SUBAPPLICATION mapping_Uebung_033 (* LED Strip Blinkende LED *)
  (* Standard: 61499-2; Description: Copyright (c) 2023 Meisterschulen am Ostbahnhof This program and the accompanying materials are made available under the terms of the Eclipse Public License 2.0 which is available at https://www.eclipse.org/legal/epl-2.0/ SPDX-License-Identifier: EPL-2.0 *)
  (* Version 1.0, 2023-10-23, Franz Höpfinger, Meisterschulen am Ostbahnhof *)
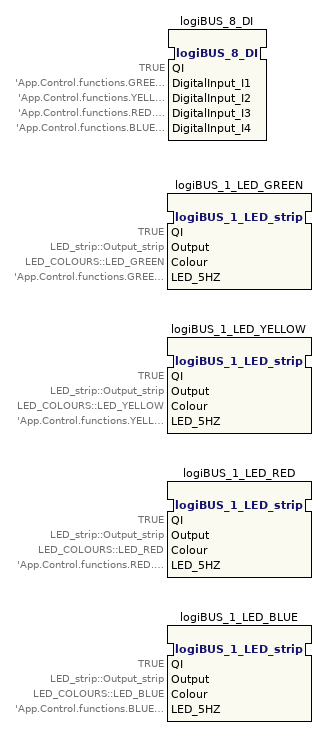
  FBS
    logiBUS_8_DI : logiBUS_8_DI(QI := TRUE, DigitalInput_I1 := 'App.Control.functions.GREEN.BUTTON', DigitalInput_I2 := 'App.Control.functions.YELLOW.BUTTON', DigitalInput_I3 := 'App.Control.functions.RED.BUTTON', DigitalInput_I4 := 'App.Control.functions.BLUE.BUTTON');
    logiBUS_1_LED_YELLOW : logiBUS_1_LED_strip(QI := TRUE, Output := LED_strip::Output_strip, Colour := LED_COLOURS::LED_YELLOW, LED_5HZ := 'App.Control.functions.YELLOW.LED');
    logiBUS_1_LED_GREEN : logiBUS_1_LED_strip(QI := TRUE, Output := LED_strip::Output_strip, Colour := LED_COLOURS::LED_GREEN, LED_5HZ := 'App.Control.functions.GREEN.LED');
    logiBUS_1_LED_RED : logiBUS_1_LED_strip(QI := TRUE, Output := LED_strip::Output_strip, Colour := LED_COLOURS::LED_RED, LED_5HZ := 'App.Control.functions.RED.LED');
    logiBUS_1_LED_BLUE : logiBUS_1_LED_strip(QI := TRUE, Output := LED_strip::Output_strip, Colour := LED_COLOURS::LED_BLUE, LED_5HZ := 'App.Control.functions.BLUE.LED');
  END_FBS
END_SUBAPPLICATION
